// TIA Portal V19 export
FUNCTION_BLOCK "A0302_Bordatrice_FB"   // FB2, LAD
TITLE = == GESTIONE DELLA STAZIONE BORDATRICE ==
// stored: MemoryReserve 100, SetENOAutomatically false
   VAR_INPUT
      AreaInterface : "AreaInterface";
      ZSI : "udt_ZoneSafetyInterface";
      DSI : "udt_DeviceSafetyInterface";
      Drive : "TAx_DriveInterface";
      DataIn : Struct
         OP : "Ax_PB";
         Sens { ExternalAccessible := 'False'; ExternalVisible := 'False'; ExternalWritable := 'False'} : Struct
            FTC_Uscita : Bool;
         END_STRUCT;
         FdBack : Struct
            ConnMotori : Bool;
            ConnAux : Bool;
         END_STRUCT;
      END_STRUCT;
      CIn { ExternalAccessible := 'False'; ExternalVisible := 'False'; ExternalWritable := 'False'} : Struct
         Manager : Struct
            Ax : "Positioning_EPOS_Machine_Manager";
            Ax_Req : Struct
               Pos0 : Bool;
               Pos1 : Bool;
               Pos2 : Bool;
               Pos3 : Bool;
            END_STRUCT;
         END_STRUCT;
         SemiAut_Pb : Bool;
         P5 : Struct
            Sollevatori : "ValveMachine_COut";
            SpintoreLong : "ValveMachine_COut";
            Sens : Struct
               FTC_Ingombro_A0301 : Bool;   // 1614BF1 - I50.7
            END_STRUCT;
         END_STRUCT;
         Rulliera : Struct
            Ax_1 : "SpeedMachine_COut";
            Centratori : "ValveMachine_COut";
            Sollevatori : "ValveMachine_COut";
            Coda : Struct
               Sens : Struct
                  FTC_Rall : Bool;   // Sensori presenza materiale banco rallentamento ingresso
                  FTC_Prox_Ing : Bool;   // Sensori presenza materiale banco limite ingresso
               END_STRUCT;
            END_STRUCT;
            Centro : Struct
               Sens : Struct
                  FTC_Centrale : Bool;   // 2010BF1 - I50.2
               END_STRUCT;
            END_STRUCT;
         END_STRUCT;
         CarroPareggCoda : Struct
            Ax : "Positioning_DOL_Machine_COut";
            Bloccaggio : "ValveMachine_COut";
            BattutaVerticale : "ValveMachine_COut";
            PareggiatoreLongitudinale : "ValveMachine_COut";
            Sens : Struct
               FTC_Ingombro_In : Bool;   // 2012BF1 - I50.0
               FTC_Ingombro_Out : Bool;   // 2012BF2 - I50.1
               PresenzaMat : Bool;   // FC presenza materiale agganciato lato paregg coda
               PosPareggLong : Struct
                  Value : LReal;
                  CheckMeasure : Bool;
                  Standstill : Bool;
               END_STRUCT;
            END_STRUCT;
         END_STRUCT;
         CarroPareggTesta : Struct
            Ax : "Positioning_DOL_Machine_COut";
            Bloccaggio : "ValveMachine_COut";
            Centraggio : "ValveMachine_COut";
            Sollevatore : "ValveMachine_COut";
            Sens : Struct
               FTC1_Rall : Bool;   // 2010BF2 - I50.3
               FTC2_Prox_Ls : Bool;   // 2010BF3 - I50.4
               PresenzaMat : Bool;   // FC presenza materiale agganciato lato paregg testa
            END_STRUCT;
         END_STRUCT;
         Attrezzaggio : Struct
            CarriParegg : Struct
               Ready : Bool;
            END_STRUCT;
            BordRegFormato : Struct
               Ready : Bool;
            END_STRUCT;
         END_STRUCT;
      END_STRUCT;
      Config : Struct
         Ax : "Positioning_EPOS_Machine_Config_NEW";
         Measure : Struct
            K1_CarroPost : LReal;   // K1: Misura tra carro di coda e sensore applicato per controllo ingombro pezzo con carro giù
            K2_BancoIngresso : LReal;   // K2: Misura interasse tra lo 0 al centro del banco e la FTC all'uscita della Bordatrice
         END_STRUCT;
      END_STRUCT;
      HWID_TEL111 : HW_SUBMODULE;
   END_VAR
   VAR_OUTPUT
      MachineInterface { ExternalAccessible := 'False'; ExternalVisible := 'False'; ExternalWritable := 'False'} : "MachineInterface";
      DataOut : "Positioning_EPOS_Machine_DataOut";
      COut : Struct
         Ax : "Positioning_EPOS_Machine_COut";
         Ax_VelOveride : Struct
            Enable : Bool;
            Value : Real;
         END_STRUCT;
         Sts : Struct
            PosTargetEnable : Bool;
            PosTarget_Reached : Bool;
            In_W_Pos : Bool;
            AtRest : Bool;
         END_STRUCT;
         DataOut : "Positioning_EPOS_Machine_DataOut";
      END_STRUCT;
   END_VAR
   VAR_IN_OUT
      Par : Struct
         Ax_Man : "Positioning_EPOS_Machine_Par";
         Ax_Aut : "A0301_Mach_Speed_Par";
      END_STRUCT;
      Pers_Data : Struct
         EncoderAbsolute_Preset_OK : Bool;
         Persistent_ActualPosition : LReal;
      END_STRUCT;
   END_VAR
   VAR
      Alarm : Struct
         Ax { ExternalVisible := 'False'} : "Positioning_EPOS_Machine_Alr";
         StopIngombroCarroCoda : Bool;
         ConnMotori_FdBack : Bool;
         ConnAux_FdBack : Bool;
      END_STRUCT;
      Warning : Struct
         Ax { S7_SetPoint := 'True'} : "Positioning_EPOS_Machine_Wng";
         OP_REST_MissingCnd : Bool;   // Mancanza comando arresto
         OP_WORK_MissingCnd : Bool;   // Mancanza consenso lavoro
      END_STRUCT;
      Ax { S7_SetPoint := 'True'} : "Positioning_EPOS_Machine_FB_NEW";
      ValueVelOvr { ExternalAccessible := 'False'; ExternalVisible := 'False'; ExternalWritable := 'False'} : Array[1..10] of Real;
      Sts : Struct
         ReadyForMove : Bool;   // Pronto al movimento
         OP_CanMoveFreely : Bool;
         OP_MoveToPos_Cnd : Bool;
         OP_Bwd_Cnd : Bool;
         OP_Fwd_Cnd : Bool;
         Pz_UscitaBord : Bool;   // Pezzo in uscita dalla Bordatrice
         StopBordatrice : Bool;   // Stop Bordatrice da controllo quota spazio rimanente su rulliera di coda
         StandbyBordatrice : Bool;
      END_STRUCT;
      Ctrl : Struct
         Bordatrice : Struct
            OP_Bwd_Man : Bool;
            OP_Fwd_Man : Bool;
            OP_Bwd_Aut : Bool;
            OP_Fwd_Aut : Bool;
            OP_Bwd_Run : Bool;
            OP_Fwd_Run : Bool;
            OP_MoveToPos : Bool;
         END_STRUCT;
         Value : Struct
            Ax_TargetLongPos { ExternalAccessible := 'False'; ExternalVisible := 'False'; ExternalWritable := 'False'} : LReal;
            QuotaInizioUscita : LReal;
            QuotaFineUscita : LReal;
            PosTarget : LReal;
            QuotaRimanenteRullieraCoda : LReal;
         END_STRUCT;
         PosTargetEnable : Bool;
      END_STRUCT;
      HMI : Struct
         Pos : LReal;
      END_STRUCT;
      AUX : Struct
         Bordatrice : Struct
            OP_Bwd_Minus_PB : Bool;
            OP_Fwd_Plus_PB : Bool;
            OP_MoveToPos_PB { ExternalAccessible := 'False'; ExternalVisible := 'False'; ExternalWritable := 'False'} : Bool;
         END_STRUCT;
         Measure : Struct
            QuotaInizio : Bool;
            QuotaFine : Bool;
         END_STRUCT;
      END_STRUCT;
      IEC_FTC_UscitaBordatrice : Struct
         TON_Delay : IEC_TIMER;
         TOF_Delay { S7_SetPoint := 'True'} : IEC_TIMER;
         FTC_On { S7_SetPoint := 'True'} : Bool;
      END_STRUCT;
      IEC_StandbyBordatrice : IEC_TIMER;
      BTrk_Item : Struct
         BLean : Real;
         O_ID : DInt;
      END_STRUCT;
   END_VAR
   VAR_TEMP
      PE : Struct
         Bordatrice : Struct
            OP_Bwd_Minus_PB : Bool;
            OP_Fwd_Plus_PB : Bool;
            OP_MoveToPos_PB : Bool;
         END_STRUCT;
      END_STRUCT;
      VelOvr_Max : Real;   // Velocità max trovata
      i : Int;
      j : Int;
      CostB : LReal;
      Module : LReal;
      M_PosAPlusCostB : LReal;
      BTrk_GetData : Struct
         indx : Int;   // Se trovato tra i TODO / ENDING / OUT questo è l'indice dove sono stati prelevati i dati
         Sts : Int;   // 0 = Non Trovato; 0 = ACT; 1 = TODO; 2=ENDING; 3 = OUT
         Item : "Prod_Item_small";
      END_STRUCT;
      PositioningStop : Bool;
      NoTrk_Bordatrice : Bool;
   END_VAR
   VAR_TEMP   // added for the SCL form of the ladder/FBD networks
      _w1 : Bool;
      _w2 : Bool;
      _w3 : Bool;
      _w4 : Bool;
      _w5 : Bool;
      _w6 : Bool;
   END_VAR
BEGIN

REGION Network 1 (SCL): Reset allarmi
   IF #AreaInterface.RstAlarms THEN
       #Alarm.StopIngombroCarroCoda := FALSE;

       IF #DataIn.FdBack.ConnMotori AND #Alarm.ConnMotori_FdBack THEN
           #Alarm.ConnMotori_FdBack := FALSE;
       END_IF;

       IF #DataIn.FdBack.ConnAux AND #Alarm.ConnAux_FdBack THEN
           #Alarm.ConnAux_FdBack := FALSE;
       END_IF;
   END_IF;
   //
END_REGION

REGION Network 2: Controllo FdBack connettori
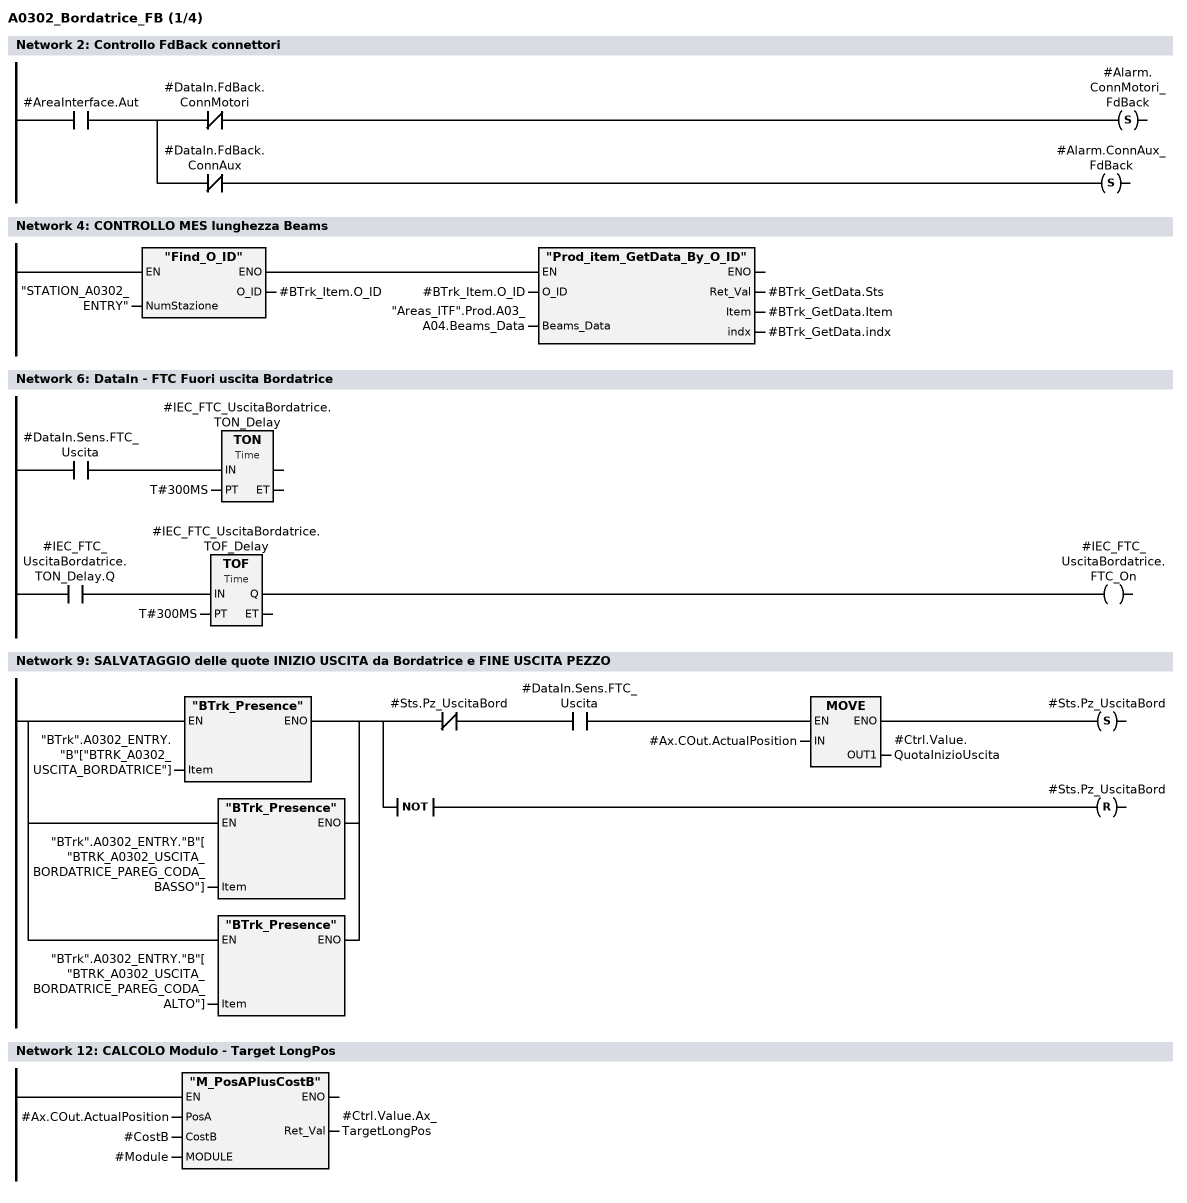
   RUNG wire#powerrail
      Contact( #AreaInterface.Aut )
      wire#w1
      I_Contact( #DataIn.FdBack.ConnMotori )
      S_Coil( #Alarm.ConnMotori_FdBack )
   END_RUNG
   RUNG wire#w1
      I_Contact( #DataIn.FdBack.ConnAux )
      S_Coil( #Alarm.ConnAux_FdBack )
   END_RUNG
   // the same network as SCL:
   IF #AreaInterface.Aut AND NOT #DataIn.FdBack.ConnMotori THEN #Alarm.ConnMotori_FdBack := TRUE; END_IF;
   IF #AreaInterface.Aut AND NOT #DataIn.FdBack.ConnAux THEN #Alarm.ConnAux_FdBack := TRUE; END_IF;
END_REGION

REGION Network 3: <+>
END_REGION

REGION Network 4: CONTROLLO MES lunghezza Beams
   RUNG wire#powerrail
      "Find_O_ID"(NumStazione := "STATION_A0302_ENTRY", O_ID => #BTrk_Item.O_ID)
      "Prod_item_GetData_By_O_ID"(O_ID := #BTrk_Item.O_ID, Beams_Data := "Areas_ITF".Prod.A03_A04.Beams_Data, Ret_Val => #BTrk_GetData.Sts, Item => #BTrk_GetData.Item, indx => #BTrk_GetData.indx)
   END_RUNG
   // the same network as SCL:
   "Find_O_ID"(NumStazione := "STATION_A0302_ENTRY", O_ID => #BTrk_Item.O_ID, ENO => #_w1);
   IF #_w1 THEN
       #BTrk_GetData.Sts := "Prod_item_GetData_By_O_ID"(O_ID := #BTrk_Item.O_ID,
                               Beams_Data := "Areas_ITF".Prod.A03_A04.Beams_Data,
                               Item => #BTrk_GetData.Item,
                               indx => #BTrk_GetData.indx);
   END_IF;
END_REGION

REGION Network 5 (SCL): CONTROLLO TRK lunghezza Beams
   //
   FOR #j:= 1 TO "BTRK_A0302_ENTRY_ITEMS" DO
       // 
       IF "BTrk".A0302_ENTRY.B[#j].BLen_Meas <> 0 THEN
           #BTrk_Item.BLean := "BTrk".A0302_ENTRY.B[#j].BLen_Meas;
       END_IF;

   END_FOR;
END_REGION

REGION Network 6: DataIn - FTC Fuori uscita Bordatrice
   RUNG wire#powerrail
      Contact( #DataIn.Sens.FTC_Uscita )
      { S7_Templates := "time_type := Time" } #IEC_FTC_UscitaBordatrice.TON_Delay.TON(pt := T#300MS, et =>)
   END_RUNG
   RUNG wire#powerrail
      Contact( #IEC_FTC_UscitaBordatrice.TON_Delay.Q )
      { S7_Templates := "time_type := Time" } #IEC_FTC_UscitaBordatrice.TOF_Delay.TOF(pt := T#300MS, et =>)
      Coil( #IEC_FTC_UscitaBordatrice.FTC_On )
   END_RUNG
   // the same network as SCL:
   #IEC_FTC_UscitaBordatrice.TON_Delay.TON(IN := #DataIn.Sens.FTC_Uscita, PT := T#300MS);
   #IEC_FTC_UscitaBordatrice.TOF_Delay.TOF(IN := #IEC_FTC_UscitaBordatrice.TON_Delay.Q, PT := T#300MS);
   #IEC_FTC_UscitaBordatrice.FTC_On := #IEC_FTC_UscitaBordatrice.TOF_Delay.Q;
END_REGION

REGION Network 7: <<<< CALCOLI QUOTE >>>>
END_REGION

REGION Network 8: <+>
END_REGION

REGION Network 9: SALVATAGGIO delle quote INIZIO USCITA da Bordatrice e FINE USCITA PEZZO
   RUNG wire#powerrail
      "BTrk_Presence"(Item := "BTrk".A0302_ENTRY."B"["BTRK_A0302_USCITA_BORDATRICE"])
      wire#w1
      I_Contact( #Sts.Pz_UscitaBord )
      Contact( #DataIn.Sens.FTC_Uscita )
      Move(in := #Ax.COut.ActualPosition, out1 => #Ctrl.Value.QuotaInizioUscita)
      S_Coil( #Sts.Pz_UscitaBord )
   END_RUNG
   RUNG wire#powerrail
      "BTrk_Presence"(Item := "BTrk".A0302_ENTRY."B"["BTRK_A0302_USCITA_BORDATRICE_PAREG_CODA_BASSO"])
   END_RUNG wire#w1
   RUNG wire#powerrail
      "BTrk_Presence"(Item := "BTrk".A0302_ENTRY."B"["BTRK_A0302_USCITA_BORDATRICE_PAREG_CODA_ALTO"])
   END_RUNG wire#w1
   RUNG wire#w1
      Not()
      R_Coil( #Sts.Pz_UscitaBord )
   END_RUNG
   // the same network as SCL:
   "BTrk_Presence"(Item := "BTrk".A0302_ENTRY."B"["BTRK_A0302_USCITA_BORDATRICE"], ENO => #_w1);
   "BTrk_Presence"(Item := "BTrk".A0302_ENTRY."B"["BTRK_A0302_USCITA_BORDATRICE_PAREG_CODA_BASSO"], ENO => #_w2);
   "BTrk_Presence"(Item := "BTrk".A0302_ENTRY."B"["BTRK_A0302_USCITA_BORDATRICE_PAREG_CODA_ALTO"], ENO => #_w3);
   #_w4 := #_w1 OR #_w2 OR #_w3;
   IF #_w4 AND NOT #Sts.Pz_UscitaBord AND #DataIn.Sens.FTC_Uscita THEN
       #Ctrl.Value.QuotaInizioUscita := #Ax.COut.ActualPosition;
       #Sts.Pz_UscitaBord := TRUE;
   END_IF;
   IF NOT #_w4 THEN #Sts.Pz_UscitaBord := FALSE; END_IF;
END_REGION

REGION Network 10 (SCL): CALCOLO dello spazio rimanete rulliera di coda
   (*** Calcolo quota Target pezzo - Se ho il carro di coda basso il target è pari alla lunghezza del pezzo
   IF #Sts.Pz_UscitaBord THEN
       #Ctrl.Value.PosTarget := #Ctrl.Value.QuotaInizioUscita + #BTrk_Item.BLean;
    END_IF; ***)

   // Calcolo dello Spazio prima del Pareggiatore di coda quando è in posizione
   // 
   #Ctrl.Value.QuotaRimanenteRullieraCoda := ((#Config.Measure.K2_BancoIngresso - #Config.Measure.K1_CarroPost) - #CIn.CarroPareggCoda.Ax.ActualPosition - 200.0);
   //
END_REGION

REGION Network 11 (SCL): CALCOLO Posizioni Target per lavoro Bordatrice
   // ******************************************************************
   // Calcoli del modulo
   // 

   #Module := #Ax.Config.Ax.Modulo_S120_P2566 / 1000.0;
   #CostB := (#Module / 2) - 1000.0;

   // Calcolo quota Target pezzo
   // Se ho il carro di coda basso il target è pari alla lunghezza del pezzo
   // 
   IF #Sts.Pz_UscitaBord THEN

       IF #CIn.CarroPareggCoda.BattutaVerticale.Work OR NOT "A0302_Manager".Ctrl.TRK.BTrk.RulliereVode THEN

           #Ctrl.Value.PosTarget := "M_PosAPlusCostB"(PosA := #Ctrl.Value.QuotaInizioUscita, CostB := #Ctrl.Value.QuotaRimanenteRullieraCoda, MODULE := #Module);

           #COut.Sts.PosTargetEnable:=#Ctrl.PosTargetEnable := TRUE;

           // Se ho il carro di coda alto il target è superiore alla lunghezza del pezzo per arrivare in fondo alla rulliera
       ELSE

           #Ctrl.Value.PosTarget := #Ctrl.Value.Ax_TargetLongPos;
           #COut.Sts.PosTargetEnable := #Ctrl.PosTargetEnable := FALSE;

       END_IF;

   ELSE
       #Ctrl.Value.PosTarget := #Ctrl.Value.Ax_TargetLongPos;
       #COut.Sts.PosTargetEnable := #Ctrl.PosTargetEnable := FALSE;
   END_IF;
END_REGION

REGION Network 12: CALCOLO Modulo - Target LongPos
   RUNG wire#powerrail
      "M_PosAPlusCostB"(PosA := #Ax.COut.ActualPosition, CostB := #CostB, MODULE := #Module, Ret_Val => #Ctrl.Value.Ax_TargetLongPos)
   END_RUNG
   // the same network as SCL:
   #Ctrl.Value.Ax_TargetLongPos := "M_PosAPlusCostB"(PosA := #Ax.COut.ActualPosition,
                           CostB := #CostB,
                           MODULE := #Module);
END_REGION

REGION Network 13: <+>
END_REGION

REGION Network 14: [Ax] Sts - Standby Bordatrice per mancanza prodotto da lavorare
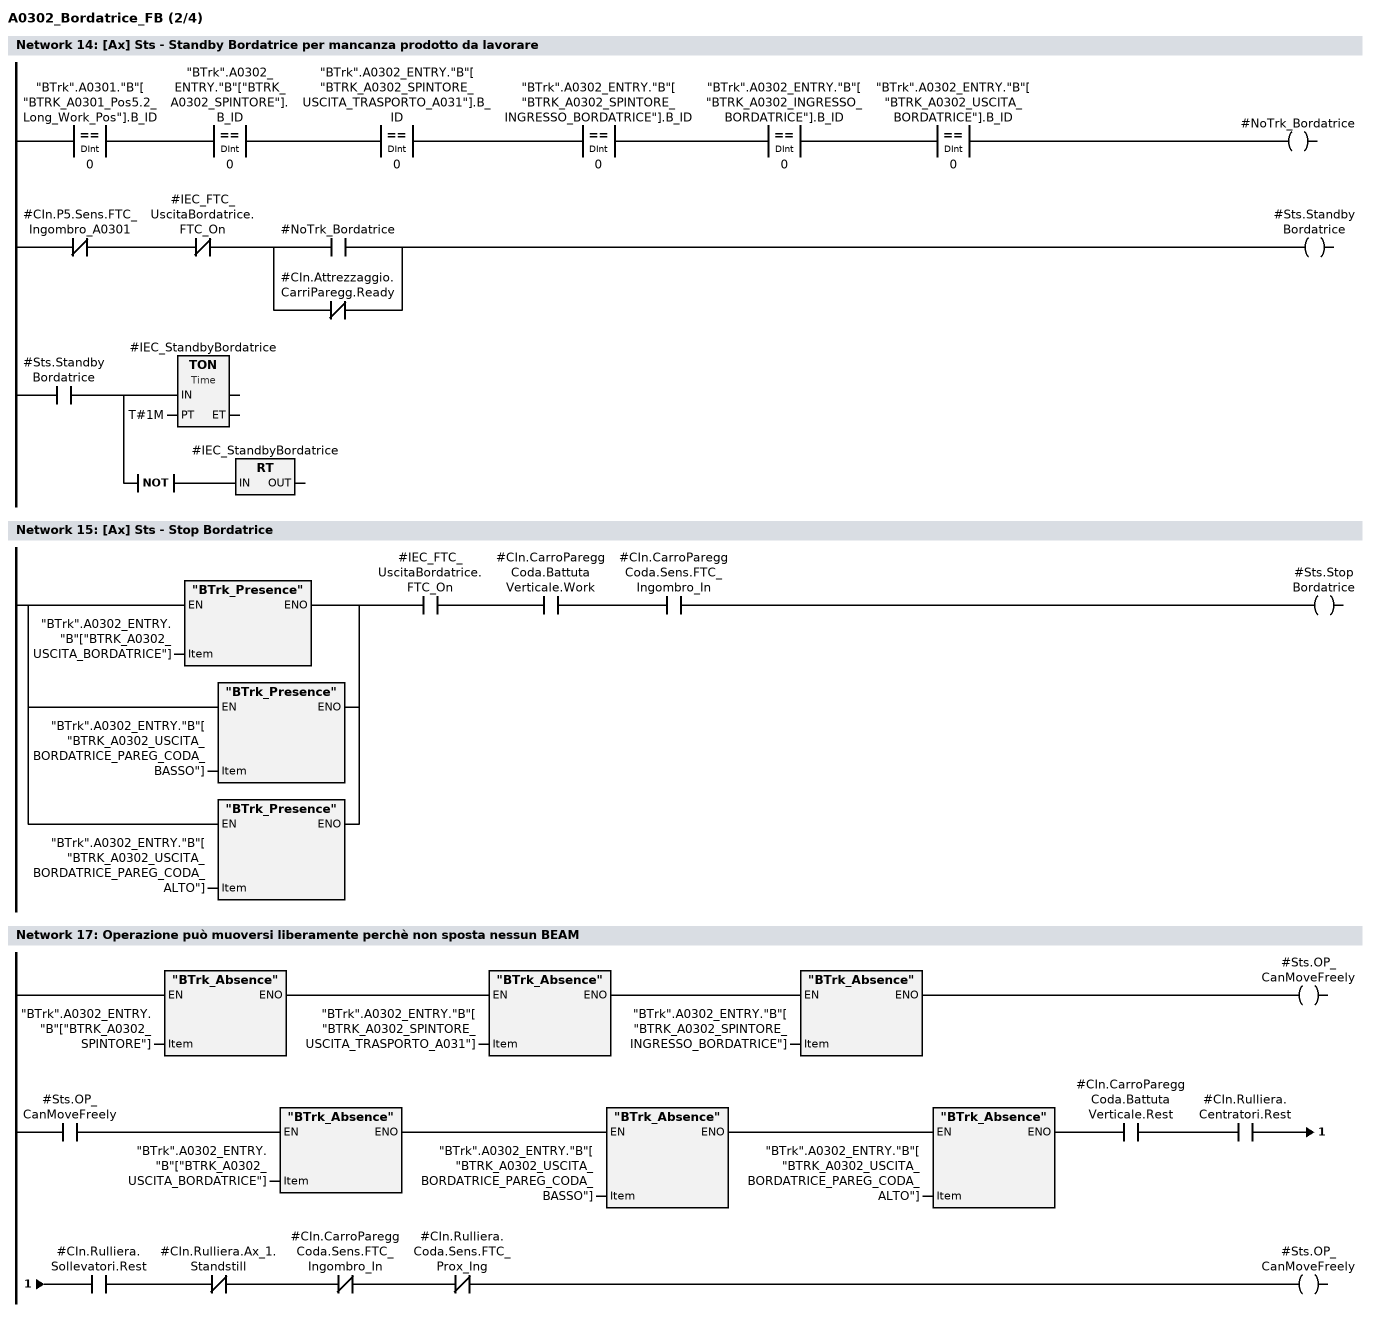
   RUNG wire#powerrail
      { S7_Templates := "SrcType := DInt" } EQ_Contact(in1 := "BTrk".A0301."B"["BTRK_A0301_Pos5.2_Long_Work_Pos"].B_ID, in2 := 0)
      { S7_Templates := "SrcType := DInt" } EQ_Contact(in1 := "BTrk".A0302_ENTRY."B"["BTRK_A0302_SPINTORE"].B_ID, in2 := 0)
      { S7_Templates := "SrcType := DInt" } EQ_Contact(in1 := "BTrk".A0302_ENTRY."B"["BTRK_A0302_SPINTORE_USCITA_TRASPORTO_A031"].B_ID, in2 := 0)
      { S7_Templates := "SrcType := DInt" } EQ_Contact(in1 := "BTrk".A0302_ENTRY."B"["BTRK_A0302_SPINTORE_INGRESSO_BORDATRICE"].B_ID, in2 := 0)
      { S7_Templates := "SrcType := DInt" } EQ_Contact(in1 := "BTrk".A0302_ENTRY."B"["BTRK_A0302_INGRESSO_BORDATRICE"].B_ID, in2 := 0)
      { S7_Templates := "SrcType := DInt" } EQ_Contact(in1 := "BTrk".A0302_ENTRY."B"["BTRK_A0302_USCITA_BORDATRICE"].B_ID, in2 := 0)
      Coil( #NoTrk_Bordatrice )
   END_RUNG
   RUNG wire#powerrail
      I_Contact( #CIn.P5.Sens.FTC_Ingombro_A0301 )
      I_Contact( #IEC_FTC_UscitaBordatrice.FTC_On )
      wire#w1
      Contact( #NoTrk_Bordatrice )
      wire#w2
      Coil( #Sts.StandbyBordatrice )
   END_RUNG
   RUNG wire#w1
      I_Contact( #CIn.Attrezzaggio.CarriParegg.Ready )
   END_RUNG wire#w2
   RUNG wire#powerrail
      Contact( #Sts.StandbyBordatrice )
      wire#w3
      { S7_Templates := "time_type := Time" } #IEC_StandbyBordatrice.TON(pt := T#1M, et =>)
   END_RUNG
   RUNG wire#w3
      Not()
      RT_Coil( #IEC_StandbyBordatrice )
   END_RUNG
   // the same network as SCL:
   #NoTrk_Bordatrice := ("BTrk".A0301."B"["BTRK_A0301_Pos5.2_Long_Work_Pos"].B_ID = 0) AND ("BTrk".A0302_ENTRY."B"["BTRK_A0302_SPINTORE"].B_ID = 0) AND ("BTrk".A0302_ENTRY."B"["BTRK_A0302_SPINTORE_USCITA_TRASPORTO_A031"].B_ID = 0) AND ("BTrk".A0302_ENTRY."B"["BTRK_A0302_SPINTORE_INGRESSO_BORDATRICE"].B_ID = 0) AND ("BTrk".A0302_ENTRY."B"["BTRK_A0302_INGRESSO_BORDATRICE"].B_ID = 0) AND ("BTrk".A0302_ENTRY."B"["BTRK_A0302_USCITA_BORDATRICE"].B_ID = 0);
   #Sts.StandbyBordatrice := NOT #CIn.P5.Sens.FTC_Ingombro_A0301 AND NOT #IEC_FTC_UscitaBordatrice.FTC_On AND (#NoTrk_Bordatrice OR NOT #CIn.Attrezzaggio.CarriParegg.Ready);
   #IEC_StandbyBordatrice.TON(IN := #Sts.StandbyBordatrice, PT := T#1M);
   IF NOT #Sts.StandbyBordatrice THEN RESET_TIMER(#IEC_StandbyBordatrice); END_IF;
END_REGION

REGION Network 15: [Ax] Sts - Stop Bordatrice
   RUNG wire#powerrail
      "BTrk_Presence"(Item := "BTrk".A0302_ENTRY."B"["BTRK_A0302_USCITA_BORDATRICE"])
      wire#w1
      Contact( #IEC_FTC_UscitaBordatrice.FTC_On )
      Contact( #CIn.CarroPareggCoda.BattutaVerticale.Work )
      Contact( #CIn.CarroPareggCoda.Sens.FTC_Ingombro_In )
      Coil( #Sts.StopBordatrice )
   END_RUNG
   RUNG wire#powerrail
      "BTrk_Presence"(Item := "BTrk".A0302_ENTRY."B"["BTRK_A0302_USCITA_BORDATRICE_PAREG_CODA_BASSO"])
   END_RUNG wire#w1
   RUNG wire#powerrail
      "BTrk_Presence"(Item := "BTrk".A0302_ENTRY."B"["BTRK_A0302_USCITA_BORDATRICE_PAREG_CODA_ALTO"])
   END_RUNG wire#w1
   // the same network as SCL:
   "BTrk_Presence"(Item := "BTrk".A0302_ENTRY."B"["BTRK_A0302_USCITA_BORDATRICE"], ENO => #_w1);
   "BTrk_Presence"(Item := "BTrk".A0302_ENTRY."B"["BTRK_A0302_USCITA_BORDATRICE_PAREG_CODA_BASSO"], ENO => #_w2);
   "BTrk_Presence"(Item := "BTrk".A0302_ENTRY."B"["BTRK_A0302_USCITA_BORDATRICE_PAREG_CODA_ALTO"], ENO => #_w3);
   #Sts.StopBordatrice := (#_w1 OR #_w2 OR #_w3) AND #IEC_FTC_UscitaBordatrice.FTC_On AND #CIn.CarroPareggCoda.BattutaVerticale.Work AND #CIn.CarroPareggCoda.Sens.FTC_Ingombro_In;
END_REGION

REGION Network 16: <+>
END_REGION

REGION Network 17: Operazione può muoversi liberamente perchè non sposta nessun BEAM
   RUNG wire#powerrail
      "BTrk_Absence"(Item := "BTrk".A0302_ENTRY."B"["BTRK_A0302_SPINTORE"])
      "BTrk_Absence"(Item := "BTrk".A0302_ENTRY."B"["BTRK_A0302_SPINTORE_USCITA_TRASPORTO_A031"])
      "BTrk_Absence"(Item := "BTrk".A0302_ENTRY."B"["BTRK_A0302_SPINTORE_INGRESSO_BORDATRICE"])
      Coil( #Sts.OP_CanMoveFreely )
   END_RUNG
   RUNG wire#powerrail
      Contact( #Sts.OP_CanMoveFreely )
      "BTrk_Absence"(Item := "BTrk".A0302_ENTRY."B"["BTRK_A0302_USCITA_BORDATRICE"])
      "BTrk_Absence"(Item := "BTrk".A0302_ENTRY."B"["BTRK_A0302_USCITA_BORDATRICE_PAREG_CODA_BASSO"])
      "BTrk_Absence"(Item := "BTrk".A0302_ENTRY."B"["BTRK_A0302_USCITA_BORDATRICE_PAREG_CODA_ALTO"])
      Contact( #CIn.CarroPareggCoda.BattutaVerticale.Rest )
      Contact( #CIn.Rulliera.Centratori.Rest )
      Contact( #CIn.Rulliera.Sollevatori.Rest )
      I_Contact( #CIn.Rulliera.Ax_1.Standstill )
      I_Contact( #CIn.CarroPareggCoda.Sens.FTC_Ingombro_In )
      I_Contact( #CIn.Rulliera.Coda.Sens.FTC_Prox_Ing )
      Coil( #Sts.OP_CanMoveFreely )
   END_RUNG
   // the same network as SCL:
   "BTrk_Absence"(Item := "BTrk".A0302_ENTRY."B"["BTRK_A0302_SPINTORE"], ENO => #_w1);
   "BTrk_Absence"(EN := #_w1,
                  Item := "BTrk".A0302_ENTRY."B"["BTRK_A0302_SPINTORE_USCITA_TRASPORTO_A031"],
                  ENO => #_w2);
   "BTrk_Absence"(EN := #_w2,
                  Item := "BTrk".A0302_ENTRY."B"["BTRK_A0302_SPINTORE_INGRESSO_BORDATRICE"],
                  ENO => #_w3);
   #Sts.OP_CanMoveFreely := #_w3;
   "BTrk_Absence"(EN := #Sts.OP_CanMoveFreely,
                  Item := "BTrk".A0302_ENTRY."B"["BTRK_A0302_USCITA_BORDATRICE"],
                  ENO => #_w4);
   "BTrk_Absence"(EN := #_w4,
                  Item := "BTrk".A0302_ENTRY."B"["BTRK_A0302_USCITA_BORDATRICE_PAREG_CODA_BASSO"],
                  ENO => #_w5);
   "BTrk_Absence"(EN := #_w5,
                  Item := "BTrk".A0302_ENTRY."B"["BTRK_A0302_USCITA_BORDATRICE_PAREG_CODA_ALTO"],
                  ENO => #_w6);
   #Sts.OP_CanMoveFreely := #_w6 AND #CIn.CarroPareggCoda.BattutaVerticale.Rest AND #CIn.Rulliera.Centratori.Rest AND #CIn.Rulliera.Sollevatori.Rest AND NOT #CIn.Rulliera.Ax_1.Standstill AND NOT #CIn.CarroPareggCoda.Sens.FTC_Ingombro_In AND NOT #CIn.Rulliera.Coda.Sens.FTC_Prox_Ing;
END_REGION

REGION Network 18: Comando Operazione Lavoro (AUT)
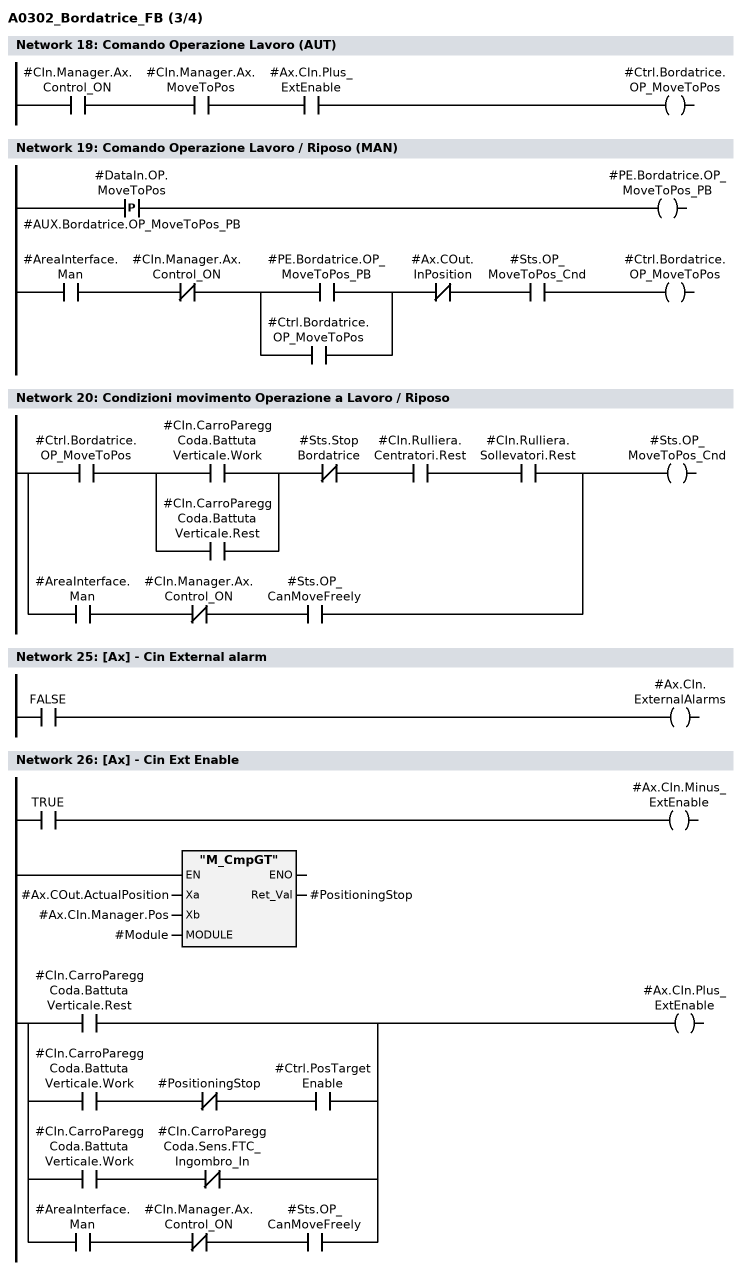
   RUNG wire#powerrail
      Contact( #CIn.Manager.Ax.Control_ON )
      Contact( #CIn.Manager.Ax.MoveToPos )
      Contact( #Ax.CIn.Plus_ExtEnable )
      Coil( #Ctrl.Bordatrice.OP_MoveToPos )
   END_RUNG
   // the same network as SCL:
   #Ctrl.Bordatrice.OP_MoveToPos := #CIn.Manager.Ax.Control_ON AND #CIn.Manager.Ax.MoveToPos AND #Ax.CIn.Plus_ExtEnable;
END_REGION

REGION Network 19: Comando Operazione Lavoro / Riposo (MAN)
   RUNG wire#powerrail
      P_Contact(operand := #DataIn.OP.MoveToPos, bit := #AUX.Bordatrice.OP_MoveToPos_PB)
      Coil( #PE.Bordatrice.OP_MoveToPos_PB )
   END_RUNG
   RUNG wire#powerrail
      Contact( #AreaInterface.Man )
      I_Contact( #CIn.Manager.Ax.Control_ON )
      wire#w1
      Contact( #PE.Bordatrice.OP_MoveToPos_PB )
      wire#w2
      I_Contact( #Ax.COut.InPosition )
      Contact( #Sts.OP_MoveToPos_Cnd )
      Coil( #Ctrl.Bordatrice.OP_MoveToPos )
   END_RUNG
   RUNG wire#w1
      Contact( #Ctrl.Bordatrice.OP_MoveToPos )
   END_RUNG wire#w2
   // the same network as SCL:
   #_w1 := #DataIn.OP.MoveToPos AND NOT #AUX.Bordatrice.OP_MoveToPos_PB;   // rising edge of #DataIn.OP.MoveToPos
   #AUX.Bordatrice.OP_MoveToPos_PB := #DataIn.OP.MoveToPos;
   #PE.Bordatrice.OP_MoveToPos_PB := #_w1;
   #Ctrl.Bordatrice.OP_MoveToPos := #AreaInterface.Man AND NOT #CIn.Manager.Ax.Control_ON AND (#PE.Bordatrice.OP_MoveToPos_PB OR #Ctrl.Bordatrice.OP_MoveToPos) AND NOT #Ax.COut.InPosition AND #Sts.OP_MoveToPos_Cnd;
END_REGION

REGION Network 20: Condizioni movimento Operazione a Lavoro / Riposo
   RUNG wire#powerrail
      Contact( #Ctrl.Bordatrice.OP_MoveToPos )
      wire#w1
      Contact( #CIn.CarroPareggCoda.BattutaVerticale.Work )
      wire#w2
      I_Contact( #Sts.StopBordatrice )
      Contact( #CIn.Rulliera.Centratori.Rest )
      Contact( #CIn.Rulliera.Sollevatori.Rest )
      wire#w3
      Coil( #Sts.OP_MoveToPos_Cnd )
   END_RUNG
   RUNG wire#w1
      Contact( #CIn.CarroPareggCoda.BattutaVerticale.Rest )
   END_RUNG wire#w2
   RUNG wire#powerrail
      Contact( #AreaInterface.Man )
      I_Contact( #CIn.Manager.Ax.Control_ON )
      Contact( #Sts.OP_CanMoveFreely )
   END_RUNG wire#w3
   // the same network as SCL:
   #Sts.OP_MoveToPos_Cnd := (#Ctrl.Bordatrice.OP_MoveToPos AND (#CIn.CarroPareggCoda.BattutaVerticale.Work OR #CIn.CarroPareggCoda.BattutaVerticale.Rest) AND NOT #Sts.StopBordatrice AND #CIn.Rulliera.Centratori.Rest AND #CIn.Rulliera.Sollevatori.Rest) OR (#AreaInterface.Man AND NOT #CIn.Manager.Ax.Control_ON AND #Sts.OP_CanMoveFreely);
END_REGION

REGION Network 21: <+>
END_REGION

REGION Network 22 (SCL): RIFERIMENTI [AX] - Positioning Manager
   // ******************************************************************************************
   REGION // TRASFERIMENTO DELLE RAMPE

       // Rampe in Manuale
       IF #AreaInterface.Man AND NOT #CIn.SemiAut_Pb THEN
           #Ax.Ctrl.Vel := #Par.Ax_Man.Man_Vel;
           #Ax.CIn.Manager.Acc := #Par.Ax_Man.Man_Acc;
           #Ax.CIn.Manager.Dec := #Par.Ax_Man.Man_Dec;
       END_IF;
   END_REGION

   // ******************************************************************************************
   REGION // // CALCOLO DELLA VELOCITA' TRASFERITA DALL'IMPIANTO IN BASE ALLA LUNGHEZZA DEL PEZZO

       // Inizializzo variabile di appoggio controllo overide massimo a un valore basso rispetto setpoint
       IF "Sys".AuxFirstPLCCycle THEN
           #VelOvr_Max := 100.0;
       END_IF;

       // Rallentamento Bordatrice con sensori
      (* 
       // Trasferisco velocità di rallentamento se ho posizionamento corto su pareggiatore di coda e raggiungo i sensori di rallentamento
       IF #Ax.#CIn.Manager.Control_ON AND #CIn.Manager.Ax.MoveToPos AND #CIn.CarroPareggCoda.BattutaVerticale.Work
           AND (#CIn.Rulliera.Coda.Sens.FTC_Rall OR #CIn.Rulliera.Coda.Sens.FTC_Prox_Ing) THEN
           #VelOvr_Max := 500.0;
       END_IF;

       // Trasferisco velocità di rallentamento se ho posizionamento lungo su pareggiatore di testa e raggiungo i sensori di rallentamento
       IF #CIn.Manager.Ax.MoveToPos AND #CIn.CarroPareggCoda.BattutaVerticale.Rest AND #CIn.Rulliera.Centro.Sens.FTC_Centrale
           AND (#CIn.CarroPareggTesta.Sens.FTC1_Rall OR #CIn.CarroPareggTesta.Sens.FTC2_Prox_Ls) THEN
           #VelOvr_Max := 500.0;
       END_IF;
       *)

       // Trasferisco le varibili su un array
       #ValueVelOvr[1] := "PPrf_MAIN".ON_WORK.A0301_A0302.Bordatrice.VelOvr_PLen_UpTo_1000;
       #ValueVelOvr[2] := "PPrf_MAIN".ON_WORK.A0301_A0302.Bordatrice.VelOvr_PLen_UpTo_1500;
       #ValueVelOvr[3] := "PPrf_MAIN".ON_WORK.A0301_A0302.Bordatrice.VelOvr_PLen_UpTo_2000;
       #ValueVelOvr[4] := "PPrf_MAIN".ON_WORK.A0301_A0302.Bordatrice.VelOvr_PLen_UpTo_2500;
       #ValueVelOvr[5] := "PPrf_MAIN".ON_WORK.A0301_A0302.Bordatrice.VelOvr_PLen_UpTo_3000;
       #ValueVelOvr[6] := "PPrf_MAIN".ON_WORK.A0301_A0302.Bordatrice.VelOvr_PLen_UpTo_3500;
       #ValueVelOvr[7] := "PPrf_MAIN".ON_WORK.A0301_A0302.Bordatrice.VelOvr_PLen_UpTo_4000;
       #ValueVelOvr[8] := "PPrf_MAIN".ON_WORK.A0301_A0302.Bordatrice.VelOvr_PLen_UpTo_4500;
       #ValueVelOvr[9] := "PPrf_MAIN".ON_WORK.A0301_A0302.Bordatrice.VelOvr_PLen_UpTo_5000;
       #ValueVelOvr[10] := "PPrf_MAIN".ON_WORK.A0301_A0302.Bordatrice.VelOvr_PLen_UpTo_5500;

       // Ciclo per verificare la variabile maggiore per prenderla in lavoro
       FOR #i := 1 TO 10 DO
           IF #ValueVelOvr[#i] >= #VelOvr_Max THEN
               #VelOvr_Max := #ValueVelOvr[#i];
           END_IF;
       END_FOR;// 
   END_REGION ;

   IF #VelOvr_Max = 0.0 THEN
       #VelOvr_Max := 100.0;
   END_IF;

   // *****************************************************************************************
   REGION // CALCOLO DELLA VELOCITA' E TRASFERIMENTO IN BASE ALLO STATO IMPIANTO

       #Ax.CIn.VelocityOverride.Enable := TRUE;
       //
       IF #Ax.CIn.Manager.Control_ON THEN

           IF #Ax.CIn.Manager.Control_ON THEN
               // CALCOLO VELOCITA' IN BASE ALL'OVERIDE
               #Ax.CIn.VelocityOverride.Value := #VelOvr_Max;
           ELSE
               #Ax.CIn.VelocityOverride.Value := 100.0;
           END_IF;

       END_IF;
   END_REGION ;
END_REGION

REGION Network 24 (SCL): [Ax] - CIn Manger
   // TRASFERIMENTO CIn MANAGER ALLA MACCHINA
   #Ax.CIn.Manager := #CIn.Manager.Ax;

   IF NOT #Ctrl.PosTargetEnable THEN
       #Ax.CIn.Manager.Pos := #Ctrl.Value.Ax_TargetLongPos;
   ELSE
       #Ax.CIn.Manager.Pos := #Ctrl.Value.PosTarget;
   END_IF;
END_REGION

REGION Network 25: [Ax] - Cin External alarm
   RUNG wire#powerrail
      Contact( FALSE )
      Coil( #Ax.CIn.ExternalAlarms )
   END_RUNG
   // the same network as SCL:
   #Ax.CIn.ExternalAlarms := FALSE;
END_REGION

REGION Network 26: [Ax] - Cin Ext Enable
   RUNG wire#powerrail
      Contact( TRUE )
      Coil( #Ax.CIn.Minus_ExtEnable )
   END_RUNG
   RUNG wire#powerrail
      "M_CmpGT"(Xa := #Ax.COut.ActualPosition, Xb := #Ax.CIn.Manager.Pos, MODULE := #Module, Ret_Val => #PositioningStop)
   END_RUNG
   RUNG wire#powerrail
      Contact( #CIn.CarroPareggCoda.BattutaVerticale.Rest )
      wire#w1
      Coil( #Ax.CIn.Plus_ExtEnable )
   END_RUNG
   RUNG wire#powerrail
      Contact( #CIn.CarroPareggCoda.BattutaVerticale.Work )
      I_Contact( #PositioningStop )
      Contact( #Ctrl.PosTargetEnable )
   END_RUNG wire#w1
   RUNG wire#powerrail
      Contact( #CIn.CarroPareggCoda.BattutaVerticale.Work )
      I_Contact( #CIn.CarroPareggCoda.Sens.FTC_Ingombro_In )
   END_RUNG wire#w1
   RUNG wire#powerrail
      Contact( #AreaInterface.Man )
      I_Contact( #CIn.Manager.Ax.Control_ON )
      Contact( #Sts.OP_CanMoveFreely )
   END_RUNG wire#w1
   // the same network as SCL:
   #Ax.CIn.Minus_ExtEnable := TRUE;
   #PositioningStop := "M_CmpGT"(Xa := #Ax.COut.ActualPosition, Xb := #Ax.CIn.Manager.Pos, MODULE := #Module);
   #Ax.CIn.Plus_ExtEnable := #CIn.CarroPareggCoda.BattutaVerticale.Rest OR (#CIn.CarroPareggCoda.BattutaVerticale.Work AND NOT #PositioningStop AND #Ctrl.PosTargetEnable) OR (#CIn.CarroPareggCoda.BattutaVerticale.Work AND NOT #CIn.CarroPareggCoda.Sens.FTC_Ingombro_In) OR (#AreaInterface.Man AND NOT #CIn.Manager.Ax.Control_ON AND #Sts.OP_CanMoveFreely);
END_REGION

REGION Network 27: [Ax] - Positioning Manager
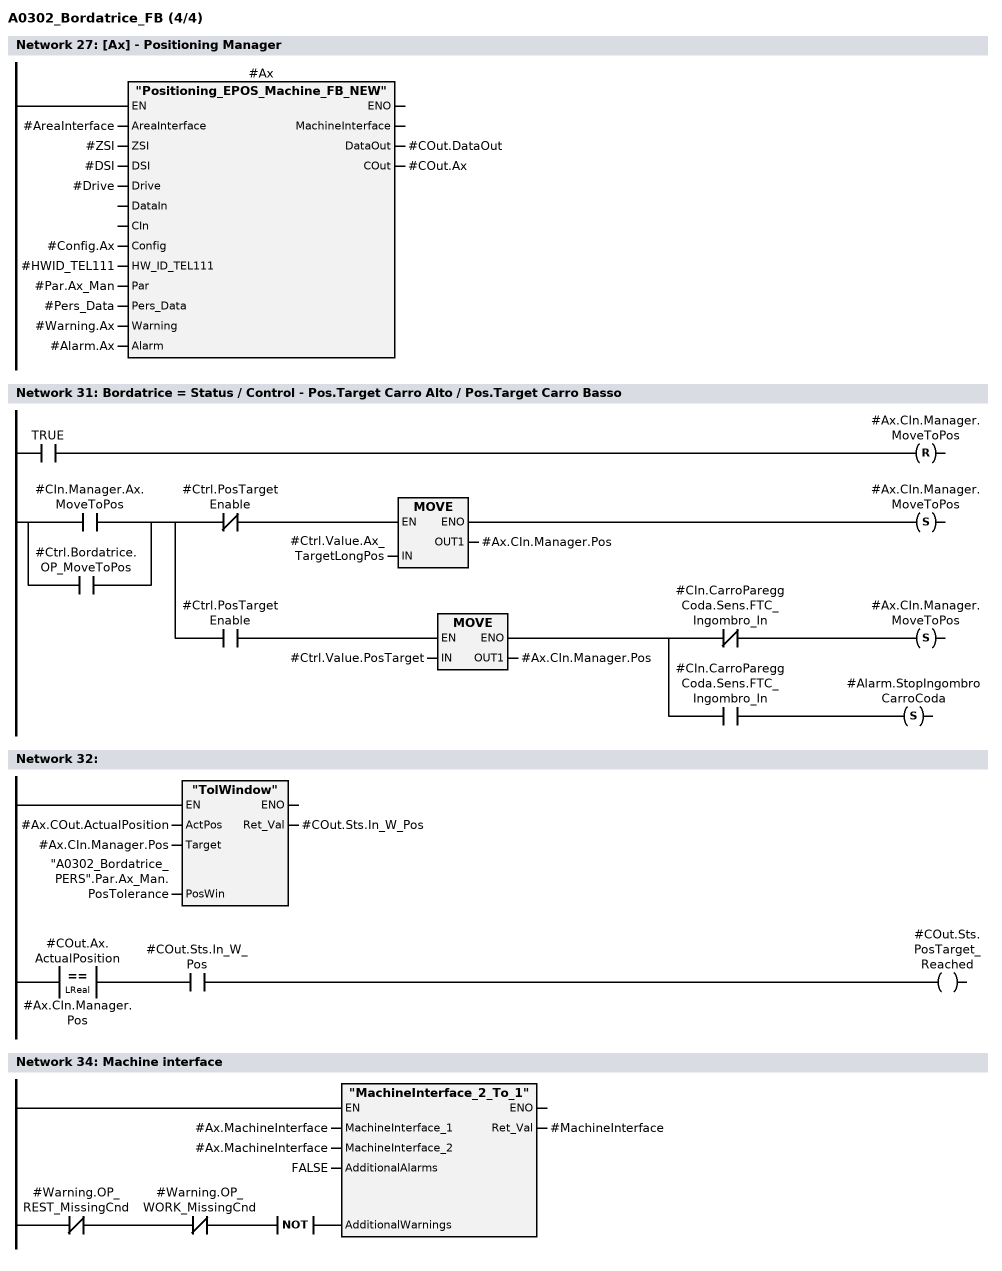
   RUNG wire#powerrail
      #Ax(AreaInterface := #AreaInterface, ZSI := #ZSI, DSI := #DSI, Drive := #Drive, DataIn :=, CIn :=, Config := #Config.Ax, HW_ID_TEL111 := #HWID_TEL111, Par := #Par.Ax_Man, Pers_Data := #Pers_Data, Warning := #Warning.Ax, Alarm := #Alarm.Ax, MachineInterface =>, DataOut => #COut.DataOut, COut => #COut.Ax)
   END_RUNG
   // the same network as SCL:
   #Ax(AreaInterface := #AreaInterface,   // "Positioning_EPOS_Machine_FB_NEW"
       ZSI := #ZSI,
       DSI := #DSI,
       Drive := #Drive,
       Config := #Config.Ax,
       HW_ID_TEL111 := #HWID_TEL111,
       Par := #Par.Ax_Man,
       Pers_Data := #Pers_Data,
       Warning := #Warning.Ax,
       Alarm := #Alarm.Ax,
       DataOut => #COut.DataOut,
       COut => #COut.Ax);
END_REGION

REGION Network 28: <+>
END_REGION

REGION Network 30: <<< CONTROLLO REQ da TRAKING E CAMBIO POS. >>>
END_REGION

REGION Network 31: Bordatrice = Status / Control - Pos.Target Carro Alto / Pos.Target Carro Basso
   RUNG wire#powerrail
      Contact( TRUE )
      R_Coil( #Ax.CIn.Manager.MoveToPos )
   END_RUNG
   RUNG wire#powerrail
      Contact( #CIn.Manager.Ax.MoveToPos )
      wire#w1
      I_Contact( #Ctrl.PosTargetEnable )
      Move(in := #Ctrl.Value.Ax_TargetLongPos, out1 => #Ax.CIn.Manager.Pos)
      S_Coil( #Ax.CIn.Manager.MoveToPos )
   END_RUNG
   RUNG wire#powerrail
      Contact( #Ctrl.Bordatrice.OP_MoveToPos )
   END_RUNG wire#w1
   RUNG wire#w1
      Contact( #Ctrl.PosTargetEnable )
      Move(in := #Ctrl.Value.PosTarget, out1 => #Ax.CIn.Manager.Pos)
      wire#w2
      I_Contact( #CIn.CarroPareggCoda.Sens.FTC_Ingombro_In )
      S_Coil( #Ax.CIn.Manager.MoveToPos )
   END_RUNG
   RUNG wire#w2
      Contact( #CIn.CarroPareggCoda.Sens.FTC_Ingombro_In )
      S_Coil( #Alarm.StopIngombroCarroCoda )
   END_RUNG
   // the same network as SCL:
   IF TRUE THEN #Ax.CIn.Manager.MoveToPos := FALSE; END_IF;
   #_w1 := #CIn.Manager.Ax.MoveToPos OR #Ctrl.Bordatrice.OP_MoveToPos;
   IF #_w1 AND NOT #Ctrl.PosTargetEnable THEN
       #Ax.CIn.Manager.Pos := #Ctrl.Value.Ax_TargetLongPos;
       #Ax.CIn.Manager.MoveToPos := TRUE;
   END_IF;
   #_w2 := #_w1 AND #Ctrl.PosTargetEnable;
   IF #_w2 THEN #Ax.CIn.Manager.Pos := #Ctrl.Value.PosTarget; END_IF;
   IF #_w2 AND NOT #CIn.CarroPareggCoda.Sens.FTC_Ingombro_In THEN #Ax.CIn.Manager.MoveToPos := TRUE; END_IF;
   IF #_w2 AND #CIn.CarroPareggCoda.Sens.FTC_Ingombro_In THEN #Alarm.StopIngombroCarroCoda := TRUE; END_IF;
END_REGION

REGION Network 32
   RUNG wire#powerrail
      "TolWindow"(ActPos := #Ax.COut.ActualPosition, Target := #Ax.CIn.Manager.Pos, PosWin := "A0302_Bordatrice_PERS".Par.Ax_Man.PosTolerance, Ret_Val => #COut.Sts.In_W_Pos)
   END_RUNG
   RUNG wire#powerrail
      { S7_Templates := "SrcType := LReal" } EQ_Contact(in1 := #COut.Ax.ActualPosition, in2 := #Ax.CIn.Manager.Pos)
      Contact( #COut.Sts.In_W_Pos )
      Coil( #COut.Sts.PosTarget_Reached )
   END_RUNG
   // the same network as SCL:
   #COut.Sts.In_W_Pos := "TolWindow"(ActPos := #Ax.COut.ActualPosition,
                           Target := #Ax.CIn.Manager.Pos,
                           PosWin := "A0302_Bordatrice_PERS".Par.Ax_Man.PosTolerance);
   #COut.Sts.PosTarget_Reached := (#COut.Ax.ActualPosition = #Ax.CIn.Manager.Pos) AND #COut.Sts.In_W_Pos;
END_REGION

REGION Network 33: << MAIN MACHINE STATUS >>
END_REGION

REGION Network 34: Machine interface
   RUNG wire#powerrail
      "MachineInterface_2_To_1"(AdditionalWarnings := wire#w1, MachineInterface_1 := #Ax.MachineInterface, MachineInterface_2 := #Ax.MachineInterface, AdditionalAlarms := FALSE, Ret_Val => #MachineInterface)
   END_RUNG
   RUNG wire#powerrail
      I_Contact( #Warning.OP_REST_MissingCnd )
      I_Contact( #Warning.OP_WORK_MissingCnd )
      Not()
   END_RUNG wire#w1
   // the same network as SCL:
   #MachineInterface := "MachineInterface_2_To_1"(MachineInterface_1 := #Ax.MachineInterface,
                           MachineInterface_2 := #Ax.MachineInterface,
                           AdditionalAlarms := FALSE,
                           AdditionalWarnings := NOT (NOT #Warning.OP_REST_MissingCnd AND NOT #Warning.OP_WORK_MissingCnd));
END_REGION
END_FUNCTION_BLOCK
